{attribute 'GeneratedUsingTerminal: EL2258-0000-0017'}
{attribute addProperty BoxType "EL2258-0000-0017"}
{attribute addProperty Id "MTO_Inputs_Channel_1AT %I*MTO_Inputs_Channel_53C09E8B6MTO_Inputs_Channel_2AT %I*MTO_Inputs_Channel_53C09E8B6MTO_Inputs_Channel_3AT %I*MTO_Inputs_Channel_53C09E8B6MTO_Inputs_Channel_4AT %I*MTO_Inputs_Channel_53C09E8B6MTO_Inputs_Channel_5AT %I*MTO_Inputs_Channel_53C09E8B6MTO_Inputs_Channel_6AT %I*MTO_Inputs_Channel_53C09E8B6MTO_Inputs_Channel_7AT %I*MTO_Inputs_Channel_53C09E8B6MTO_Inputs_Channel_8AT %I*MTO_Inputs_Channel_53C09E8B6MTO_Outputs_10x_Channel_1AT %Q*MTO_Outputs_10x_Channel_A3C0C02256MTO_Outputs_10x_Channel_2AT %Q*MTO_Outputs_10x_Channel_A3C0C02256MTO_Outputs_10x_Channel_3AT %Q*MTO_Outputs_10x_Channel_A3C0C02256MTO_Outputs_10x_Channel_4AT %Q*MTO_Outputs_10x_Channel_A3C0C02256MTO_Outputs_10x_Channel_5AT %Q*MTO_Outputs_10x_Channel_A3C0C02256MTO_Outputs_10x_Channel_6AT %Q*MTO_Outputs_10x_Channel_A3C0C02256MTO_Outputs_10x_Channel_7AT %Q*MTO_Outputs_10x_Channel_A3C0C02256MTO_Outputs_10x_Channel_8AT %Q*MTO_Outputs_10x_Channel_A3C0C02256WcStateAT %I*WcState_9091E0EB2InfoDataAT %I*InfoData_1088C70510"}
{attribute addProperty CRC "3370845153"}
{attribute addProperty Size "508"}
TYPE EL2258_C8EB03E1 EXTENDS EtcSlaveTerminalBase_947E5A46 :
STRUCT
	{attribute addProperty Name "MTO_Inputs_Channel_1"}
	MTO_Inputs_Channel_1 : MTO_Inputs_Channel_53C09E8B;
	{attribute addProperty Name "MTO_Inputs_Channel_2"}
	MTO_Inputs_Channel_2 : MTO_Inputs_Channel_53C09E8B;
	{attribute addProperty Name "MTO_Inputs_Channel_3"}
	MTO_Inputs_Channel_3 : MTO_Inputs_Channel_53C09E8B;
	{attribute addProperty Name "MTO_Inputs_Channel_4"}
	MTO_Inputs_Channel_4 : MTO_Inputs_Channel_53C09E8B;
	{attribute addProperty Name "MTO_Inputs_Channel_5"}
	MTO_Inputs_Channel_5 : MTO_Inputs_Channel_53C09E8B;
	{attribute addProperty Name "MTO_Inputs_Channel_6"}
	MTO_Inputs_Channel_6 : MTO_Inputs_Channel_53C09E8B;
	{attribute addProperty Name "MTO_Inputs_Channel_7"}
	MTO_Inputs_Channel_7 : MTO_Inputs_Channel_53C09E8B;
	{attribute addProperty Name "MTO_Inputs_Channel_8"}
	MTO_Inputs_Channel_8 : MTO_Inputs_Channel_53C09E8B;
	{attribute addProperty Name "MTO_Outputs_10x_Channel_1"}
	MTO_Outputs_10x_Channel_1 : MTO_Outputs_10x_Channel_A3C0C022;
	{attribute addProperty Name "MTO_Outputs_10x_Channel_2"}
	MTO_Outputs_10x_Channel_2 : MTO_Outputs_10x_Channel_A3C0C022;
	{attribute addProperty Name "MTO_Outputs_10x_Channel_3"}
	MTO_Outputs_10x_Channel_3 : MTO_Outputs_10x_Channel_A3C0C022;
	{attribute addProperty Name "MTO_Outputs_10x_Channel_4"}
	MTO_Outputs_10x_Channel_4 : MTO_Outputs_10x_Channel_A3C0C022;
	{attribute addProperty Name "MTO_Outputs_10x_Channel_5"}
	MTO_Outputs_10x_Channel_5 : MTO_Outputs_10x_Channel_A3C0C022;
	{attribute addProperty Name "MTO_Outputs_10x_Channel_6"}
	MTO_Outputs_10x_Channel_6 : MTO_Outputs_10x_Channel_A3C0C022;
	{attribute addProperty Name "MTO_Outputs_10x_Channel_7"}
	MTO_Outputs_10x_Channel_7 : MTO_Outputs_10x_Channel_A3C0C022;
	{attribute addProperty Name "MTO_Outputs_10x_Channel_8"}
	MTO_Outputs_10x_Channel_8 : MTO_Outputs_10x_Channel_A3C0C022;
	{attribute addProperty Name "WcState"}
	WcState : WcState_9091E0EB;
	{attribute addProperty Name "InfoData"}
	InfoData : InfoData_1088C705;
END_STRUCT
END_TYPE

(* stored: Version 1.2.0.0, ProductVersion 3.1.4024.9
   DUT EL2258_C8EB03E1: Id {c3c50af2-ce38-411b-a3a7-40e47ccda2d9} *)
